PROGRAM main
VAR
	Discharge AT %IX100.0 : bool := 1;
	I_Fill AT %IX100.1 : bool;
	Discharge_valve AT %QX100.0 : bool;
	Discharging AT %QX100.1 : bool;
	Fill_valve AT %QX100.2 : bool;
	Filling AT %QX100.3 : bool;
	Timer AT %QW100 : int;
	TOF0 : TOF;
	TOF1 : TOF;
	fill_time_to_count : time;
	discharge_time_to_count : time;
	only_dis : bool;
	only_fill : bool;
END_VAR

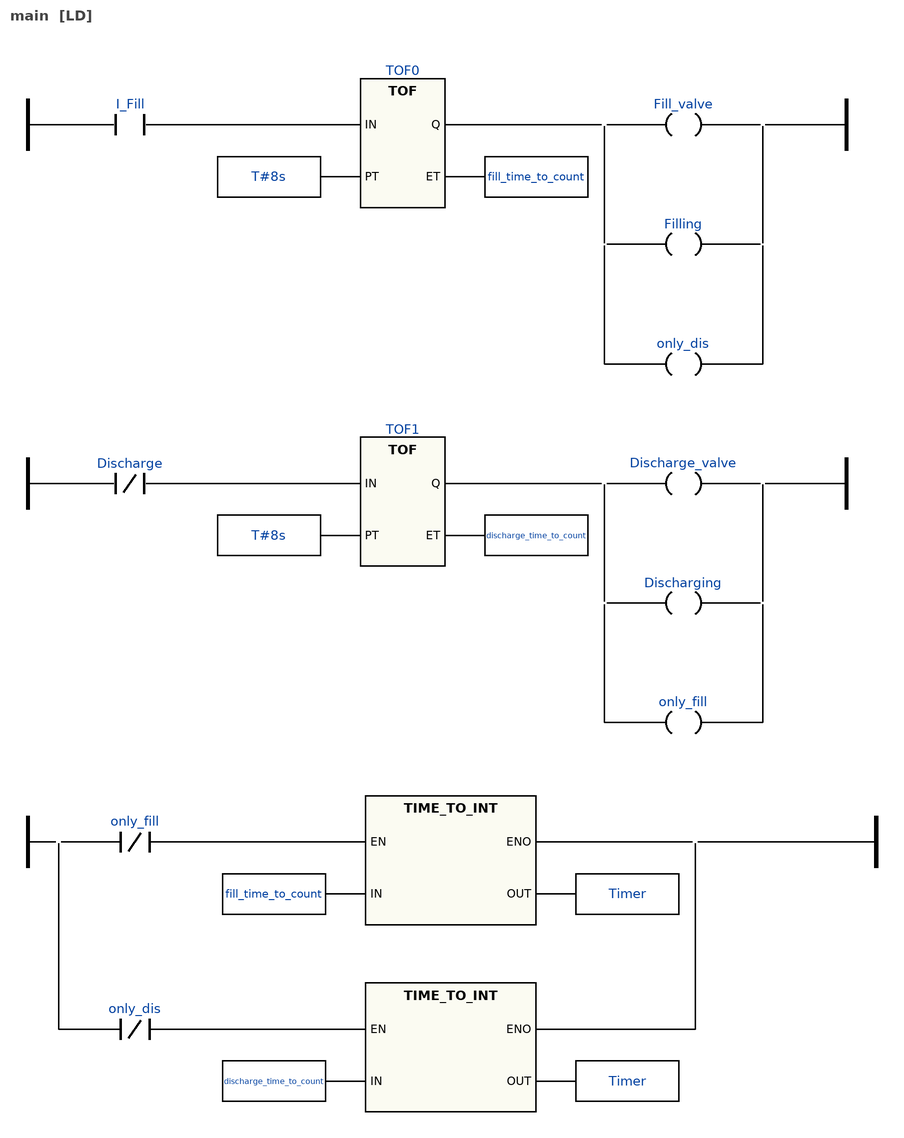
(* LD diagram, written out as Structured Text *)
TOF0(IN := I_Fill, PT := T#8s);
Fill_valve := TOF0.Q;
Filling := TOF0.Q;
only_dis := TOF0.Q;
fill_time_to_count := TOF0.ET;
TOF1(IN := NOT Discharge, PT := T#8s);
Discharge_valve := TOF1.Q;
Discharging := TOF1.Q;
only_fill := TOF1.Q;
discharge_time_to_count := TOF1.ET;
IF NOT only_fill THEN Timer := TIME_TO_INT(fill_time_to_count); END_IF;
IF NOT only_dis THEN Timer := TIME_TO_INT(discharge_time_to_count); END_IF;
END_PROGRAM
